PROGRAM MAIN
VAR
END_VAR

END_PROGRAM

(* stored: Version 1.1.0.1
   POU MAIN: Id {0184b93c-86f2-49ff-8377-c88381db76d0} *)
